Omron CX-Programmer project 疏蜞轳觇開钺祛蝼桕 (CX-Programmer 9.41)

# PLC 皖恹橄耸1: CP1E N40

## Global symbols (name address type ; comment)
0.00 BOOL  ; 原点接近
0.01 BOOL  ; 膜架上限
0.03 BOOL  ; 膜架下限
0.04 BOOL  ; 暂停
0.05 BOOL  ; 运行
0.06 BOOL  ; 急停
0.07 BOOL  ; 薄膜随动
0.08 BOOL  ; 减速接近
0.09 BOOL  ; 进料光电
0.11 BOOL  ; 货高与货到位光电
100.00 BOOL  ; 送膜转
100.01 BOOL  ; 模架下降
100.02 BOOL  ; 主机输送线转
100.04 BOOL  ; 转盘正传
100.05 BOOL  ; 转盘2段速
100.06 BOOL  ; 转盘3段速
100.07 BOOL  ; 膜架上升
101.00 BOOL  ; 夹膜
101.01 BOOL  ; 摆臂
101.02 BOOL  ; 断膜
101.03 BOOL  ; 扶膜
101.05 BOOL  ; 吹膜
101.07 BOOL  ; 送膜切换
102.04 BOOL  ; 压膜
102.05 BOOL  ; 吹摸
102.07 BOOL  ; 送膜切换
12.00 BOOL  ; 运行开始
12.01 BOOL  ; 进料光电触发位
12.02 BOOL  ; 触发运行延时
12.03 BOOL  ; 夹膜释放触发位
12.04 BOOL  ; 什么时候升到位
12.05 BOOL  ; 触发頂层计数
12.06 BOOL  ; 甚么时候下到位
12.07 BOOL  ; 底层技术开始
12.08 BOOL  ; 2段速进入位
12.09 BOOL  ; 2段速结束位
12.10 BOOL  ; 三段速进入位
12.11 BOOL  ; 停止位
12.12 BOOL  ; 摆臂触发位
12.13 BOOL  ; 触发出货
12.14 BOOL  ; 主机线停止
12.15 BOOL  ; 反复循环位
13.00 BOOL  ; 貨高光电触发位
13.01 BOOL  ; 停止膜上升
13.02 BOOL  ; 准备运行开始
13.03 BOOL  ; 运行准备完成
13.04 BOOL  ; 后送线停止
14.00 BOOL  ; 运行前回原点
14.01 BOOL  ; 运行前回下限位
15.00 BOOL  ; 包完后进3段速
15.01 BOOL  ; 包完后何时进3段速
1.00 BOOL  ; 出到位
1.01 BOOL  ; 货高与货到位光电
C001 BOOL  ; 减速计数
C002 BOOL  ; 底层设置数
C003 BOOL  ; 頂层计数
C004 BOOL  ; 往复次数设置数
C005 BOOL  ; 停止圈数
T010 BOOL  ; 运行延时
T011 BOOL  ; 货高延时
T012 BOOL  ; 压膜延时设置值
T013 BOOL  ; 夹膜设置值
T014 BOOL  ; 锻模设置值
T015 BOOL  ; 抚摸设置值
T016 BOOL  ; 出货设置值
T017 BOOL  ; 出货值加1
T018 BOOL  ; 吹膜延时
T100 BOOL  ; 货到延时
T200 BOOL  ; 模架下降延时
T202 BOOL  ; 落剪子延时
W10.00 BOOL  ; 手动后线转动
W10.01 BOOL  ; 模架上升触发位
W10.02 BOOL  ; 模架下降触发位
W10.03 BOOL  ; 主机输送线触发位
W10.04 BOOL  ; 手动夹膜
W10.05 BOOL  ; 手动转盘正传
W10.06 BOOL  ; 手动主机输送线转
W10.07 BOOL  ; 手动夹膜释放
W10.08 BOOL  ; 手动摆臂
W10.09 BOOL  ; 手动断膜
W10.10 BOOL  ; 手动抚摸
W10.11 BOOL  ; 手动膜架上升
W10.12 BOOL  ; 手动模架下降
W10.14 BOOL  ; 后线触发位
W10.15 BOOL  ; 手动压膜
W11.00 BOOL  ; 荚膜释放
W11.02 BOOL  ; 转盘正传触发位
W11.03 BOOL  ; 转盘2段速触发位
W11.04 BOOL  ; 转盘3段速触发位
W11.11 BOOL  ; 压膜
W11.12 BOOL  ; 锻模
W11.13 BOOL  ; 抚摸
W11.14 BOOL  ; 荚膜
W11.15 BOOL  ; 摆臂
W50.00 BOOL  ; 货到延时自锁
W80.00 BOOL  ; 夹膜释放
W80.01 BOOL  ; 荚膜
W80.02 BOOL  ; 吹膜

## Program 新程序1 (cyclic task 0)
Local symbols
好0 CHANNEL

### Section 段1

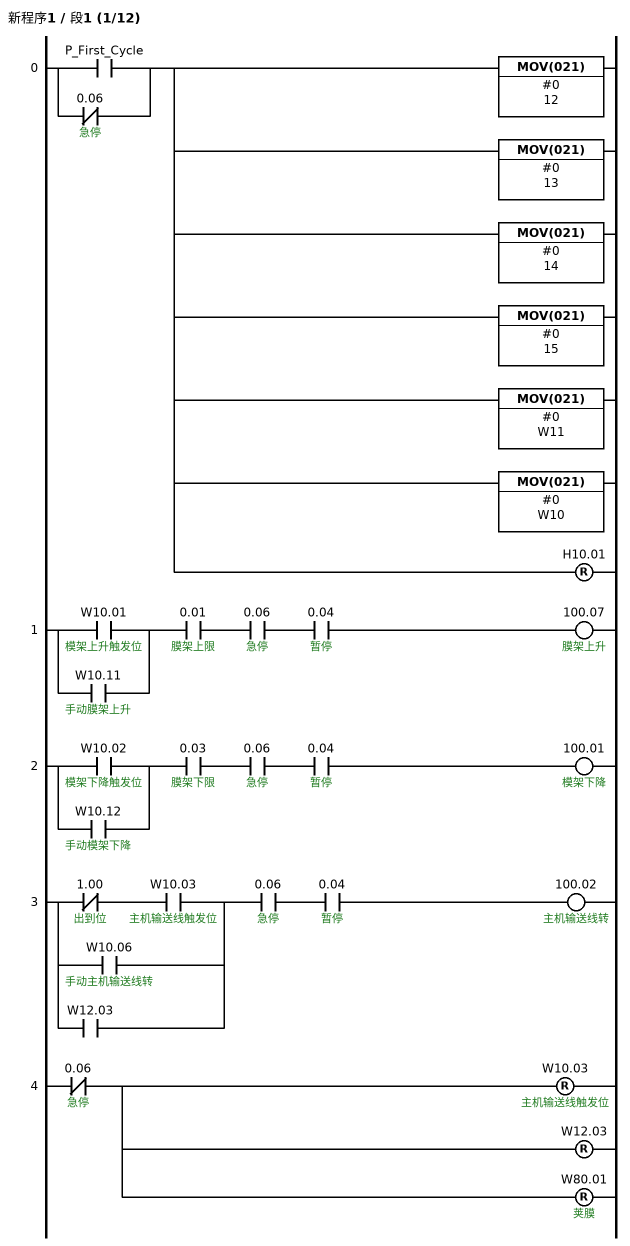
; rung 0
LD P_First_Cycle
ORNOT 0.06  ; 急停
MOV(021) #0 12
MOV(021) #0 13
MOV(021) #0 14
MOV(021) #0 15
MOV(021) #0 W11
MOV(021) #0 W10
RSET H10.01
; rung 1
LD W10.01  ; 模架上升触发位
OR W10.11  ; 手动膜架上升
AND 0.01  ; 膜架上限
AND 0.06  ; 急停
AND 0.04  ; 暂停
OUT 100.07  ; 膜架上升
; rung 2
LD W10.02  ; 模架下降触发位
OR W10.12  ; 手动模架下降
AND 0.03  ; 膜架下限
AND 0.06  ; 急停
AND 0.04  ; 暂停
OUT 100.01  ; 模架下降
; rung 3
LDNOT 1.00  ; 出到位
AND W10.03  ; 主机输送线触发位
OR W10.06  ; 手动主机输送线转
OR W12.03
AND 0.06  ; 急停
AND 0.04  ; 暂停
OUT 100.02  ; 主机输送线转
; rung 4
LDNOT 0.06  ; 急停
RSET W10.03  ; 主机输送线触发位
RSET W12.03
RSET W80.01  ; 荚膜

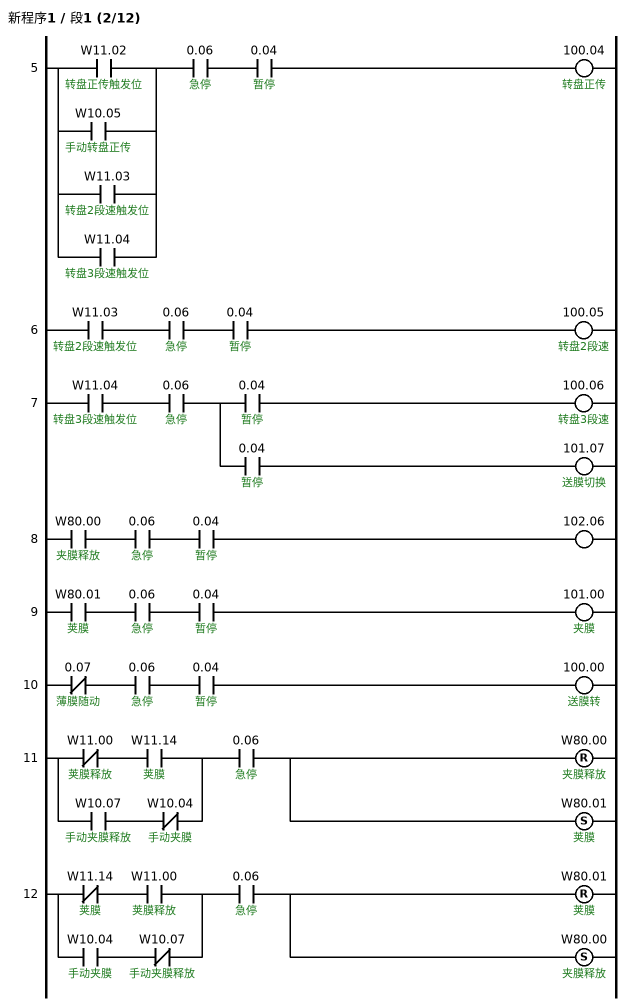
; rung 5
LD W11.02  ; 转盘正传触发位
OR W10.05  ; 手动转盘正传
OR W11.03  ; 转盘2段速触发位
OR W11.04  ; 转盘3段速触发位
AND 0.06  ; 急停
AND 0.04  ; 暂停
OUT 100.04  ; 转盘正传
; rung 6
LD W11.03  ; 转盘2段速触发位
AND 0.06  ; 急停
AND 0.04  ; 暂停
OUT 100.05  ; 转盘2段速
; rung 7
LD W11.04  ; 转盘3段速触发位
AND 0.06  ; 急停
OUT TR0
AND 0.04  ; 暂停
OUT 100.06  ; 转盘3段速
LD TR0
AND 0.04  ; 暂停
OUT 101.07  ; 送膜切换
; rung 8
LD W80.00  ; 夹膜释放
AND 0.06  ; 急停
AND 0.04  ; 暂停
OUT 102.06
; rung 9
LD W80.01  ; 荚膜
AND 0.06  ; 急停
AND 0.04  ; 暂停
OUT 101.00  ; 夹膜
; rung 10
LDNOT 0.07  ; 薄膜随动
AND 0.06  ; 急停
AND 0.04  ; 暂停
OUT 100.00  ; 送膜转
; rung 11
LDNOT W11.00  ; 荚膜释放
AND W11.14  ; 荚膜
LD W10.07  ; 手动夹膜释放
ANDNOT W10.04  ; 手动夹膜
ORLD
AND 0.06  ; 急停
RSET W80.00  ; 夹膜释放
SET W80.01  ; 荚膜
; rung 12
LDNOT W11.14  ; 荚膜
AND W11.00  ; 荚膜释放
LD W10.04  ; 手动夹膜
ANDNOT W10.07  ; 手动夹膜释放
ORLD
AND 0.06  ; 急停
RSET W80.01  ; 荚膜
SET W80.00  ; 夹膜释放

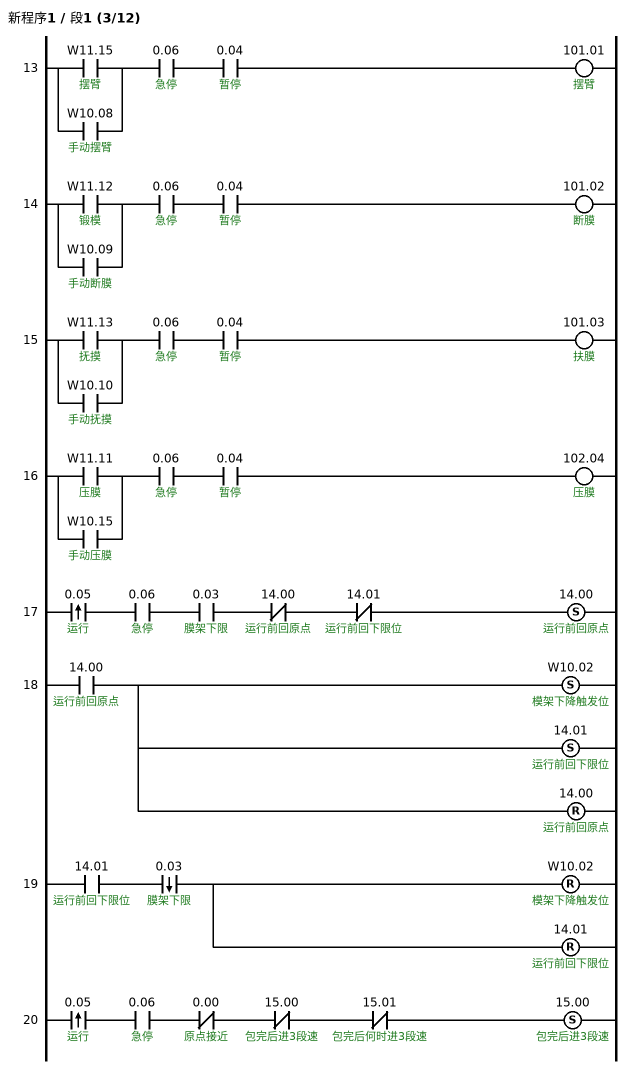
; rung 13
LD W11.15  ; 摆臂
OR W10.08  ; 手动摆臂
AND 0.06  ; 急停
AND 0.04  ; 暂停
OUT 101.01  ; 摆臂
; rung 14
LD W11.12  ; 锻模
OR W10.09  ; 手动断膜
AND 0.06  ; 急停
AND 0.04  ; 暂停
OUT 101.02  ; 断膜
; rung 15
LD W11.13  ; 抚摸
OR W10.10  ; 手动抚摸
AND 0.06  ; 急停
AND 0.04  ; 暂停
OUT 101.03  ; 扶膜
; rung 16
LD W11.11  ; 压膜
OR W10.15  ; 手动压膜
AND 0.06  ; 急停
AND 0.04  ; 暂停
OUT 102.04  ; 压膜
; rung 17
@LD 0.05  ; 运行
AND 0.06  ; 急停
AND 0.03  ; 膜架下限
ANDNOT 14.00  ; 运行前回原点
ANDNOT 14.01  ; 运行前回下限位
SET 14.00  ; 运行前回原点
; rung 18
LD 14.00  ; 运行前回原点
SET W10.02  ; 模架下降触发位
SET 14.01  ; 运行前回下限位
RSET 14.00  ; 运行前回原点
; rung 19
LD 14.01  ; 运行前回下限位
%AND 0.03  ; 膜架下限
RSET W10.02  ; 模架下降触发位
RSET 14.01  ; 运行前回下限位
; rung 20
@LD 0.05  ; 运行
AND 0.06  ; 急停
ANDNOT 0.00  ; 原点接近
ANDNOT 15.00  ; 包完后进3段速
ANDNOT 15.01  ; 包完后何时进3段速
SET 15.00  ; 包完后进3段速

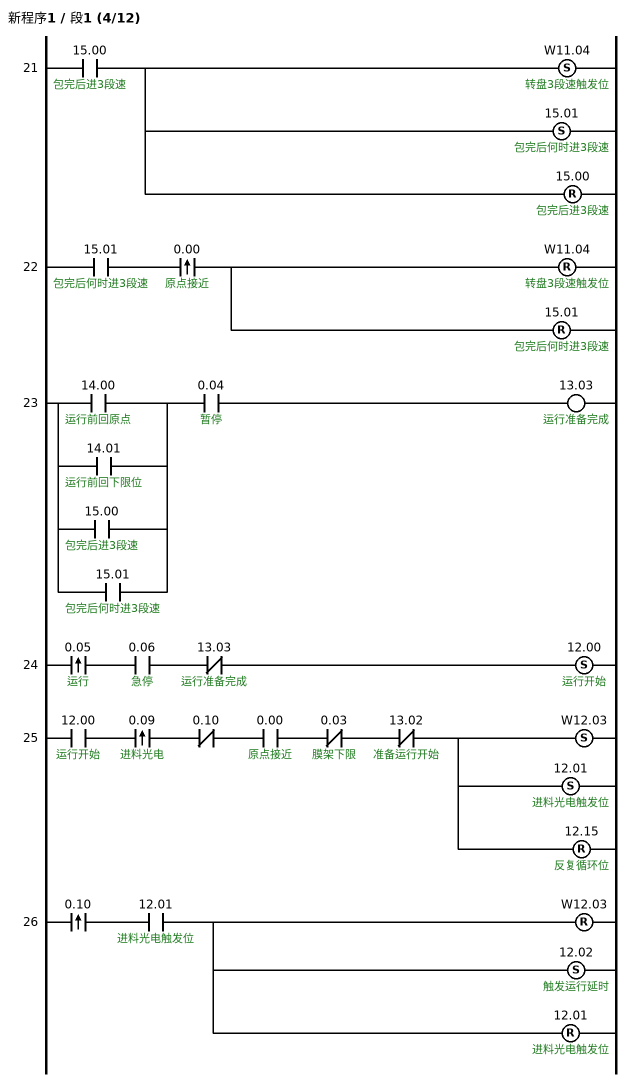
; rung 21
LD 15.00  ; 包完后进3段速
SET W11.04  ; 转盘3段速触发位
SET 15.01  ; 包完后何时进3段速
RSET 15.00  ; 包完后进3段速
; rung 22
LD 15.01  ; 包完后何时进3段速
@AND 0.00  ; 原点接近
RSET W11.04  ; 转盘3段速触发位
RSET 15.01  ; 包完后何时进3段速
; rung 23
LD 14.00  ; 运行前回原点
OR 14.01  ; 运行前回下限位
OR 15.00  ; 包完后进3段速
OR 15.01  ; 包完后何时进3段速
AND 0.04  ; 暂停
OUT 13.03  ; 运行准备完成
; rung 24
@LD 0.05  ; 运行
AND 0.06  ; 急停
ANDNOT 13.03  ; 运行准备完成
SET 12.00  ; 运行开始
; rung 25
LD 12.00  ; 运行开始
@AND 0.09  ; 进料光电
ANDNOT 0.10
AND 0.00  ; 原点接近
ANDNOT 0.03  ; 膜架下限
ANDNOT 13.02  ; 准备运行开始
SET W12.03
SET 12.01  ; 进料光电触发位
RSET 12.15  ; 反复循环位
; rung 26
@LD 0.10
AND 12.01  ; 进料光电触发位
RSET W12.03
SET 12.02  ; 触发运行延时
RSET 12.01  ; 进料光电触发位

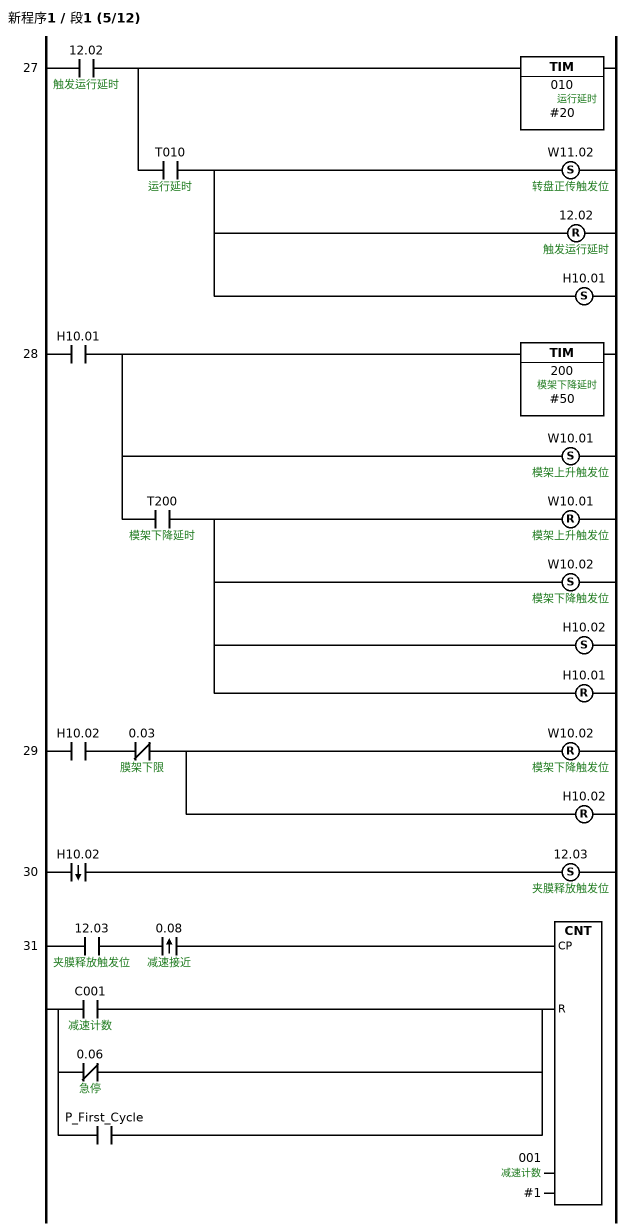
; rung 27
LD 12.02  ; 触发运行延时
TIM 010 #20  ; 运行延时
AND T010  ; 运行延时
SET W11.02  ; 转盘正传触发位
RSET 12.02  ; 触发运行延时
SET H10.01
; rung 28
LD H10.01
TIM 200 #50  ; 模架下降延时
SET W10.01  ; 模架上升触发位
AND T200  ; 模架下降延时
RSET W10.01  ; 模架上升触发位
SET W10.02  ; 模架下降触发位
SET H10.02
RSET H10.01
; rung 29
LD H10.02
ANDNOT 0.03  ; 膜架下限
RSET W10.02  ; 模架下降触发位
RSET H10.02
; rung 30
%LD H10.02
SET 12.03  ; 夹膜释放触发位
; rung 31
LD 12.03  ; 夹膜释放触发位
@AND 0.08  ; 减速接近
LD C001  ; 减速计数
ORNOT 0.06  ; 急停
OR P_First_Cycle
CNT 001 #1  ; 减速计数

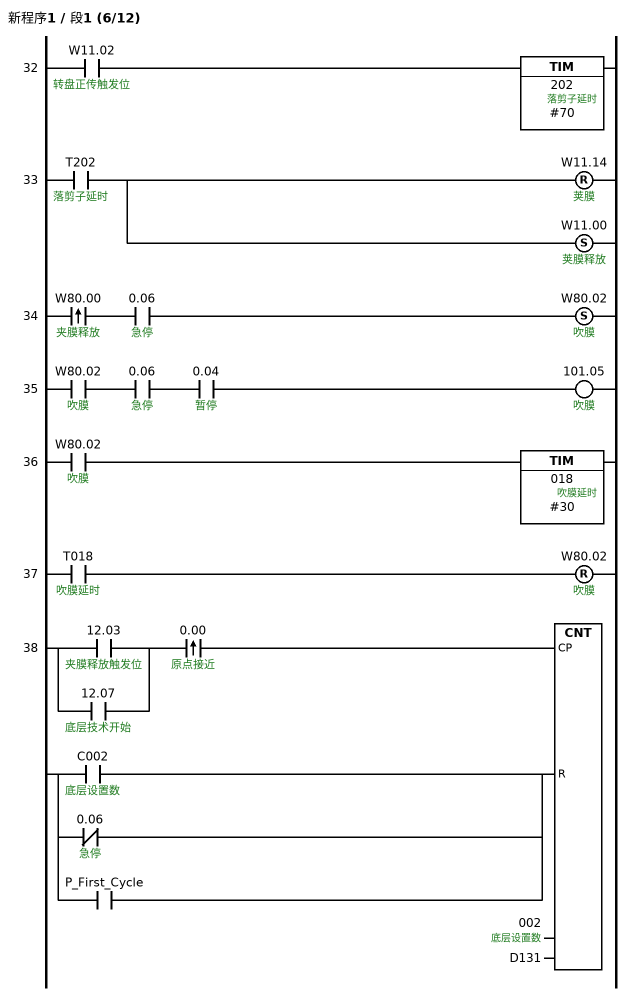
; rung 32
LD W11.02  ; 转盘正传触发位
TIM 202 #70  ; 落剪子延时
; rung 33
LD T202  ; 落剪子延时
RSET W11.14  ; 荚膜
SET W11.00  ; 荚膜释放
; rung 34
@LD W80.00  ; 夹膜释放
AND 0.06  ; 急停
SET W80.02  ; 吹膜
; rung 35
LD W80.02  ; 吹膜
AND 0.06  ; 急停
AND 0.04  ; 暂停
OUT 101.05  ; 吹膜
; rung 36
LD W80.02  ; 吹膜
TIM 018 #30  ; 吹膜延时
; rung 37
LD T018  ; 吹膜延时
RSET W80.02  ; 吹膜
; rung 38
LD 12.03  ; 夹膜释放触发位
OR 12.07  ; 底层技术开始
@AND 0.00  ; 原点接近
LD C002  ; 底层设置数
ORNOT 0.06  ; 急停
OR P_First_Cycle
CNT 002 D131  ; 底层设置数

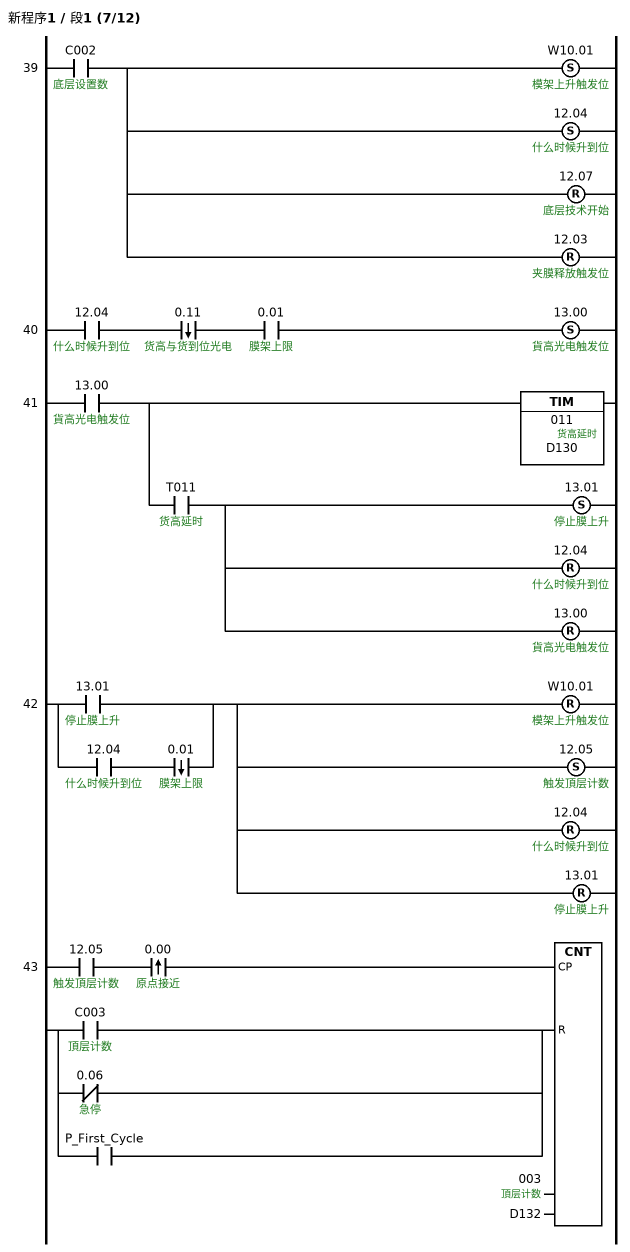
; rung 39
LD C002  ; 底层设置数
SET W10.01  ; 模架上升触发位
SET 12.04  ; 什么时候升到位
RSET 12.07  ; 底层技术开始
RSET 12.03  ; 夹膜释放触发位
; rung 40
LD 12.04  ; 什么时候升到位
%AND 0.11  ; 货高与货到位光电
AND 0.01  ; 膜架上限
SET 13.00  ; 貨高光电触发位
; rung 41
LD 13.00  ; 貨高光电触发位
TIM 011 D130  ; 货高延时
AND T011  ; 货高延时
SET 13.01  ; 停止膜上升
RSET 12.04  ; 什么时候升到位
RSET 13.00  ; 貨高光电触发位
; rung 42
LD 13.01  ; 停止膜上升
LD 12.04  ; 什么时候升到位
%AND 0.01  ; 膜架上限
ORLD
RSET W10.01  ; 模架上升触发位
SET 12.05  ; 触发頂层计数
RSET 12.04  ; 什么时候升到位
RSET 13.01  ; 停止膜上升
; rung 43
LD 12.05  ; 触发頂层计数
@AND 0.00  ; 原点接近
LD C003  ; 頂层计数
ORNOT 0.06  ; 急停
OR P_First_Cycle
CNT 003 D132  ; 頂层计数

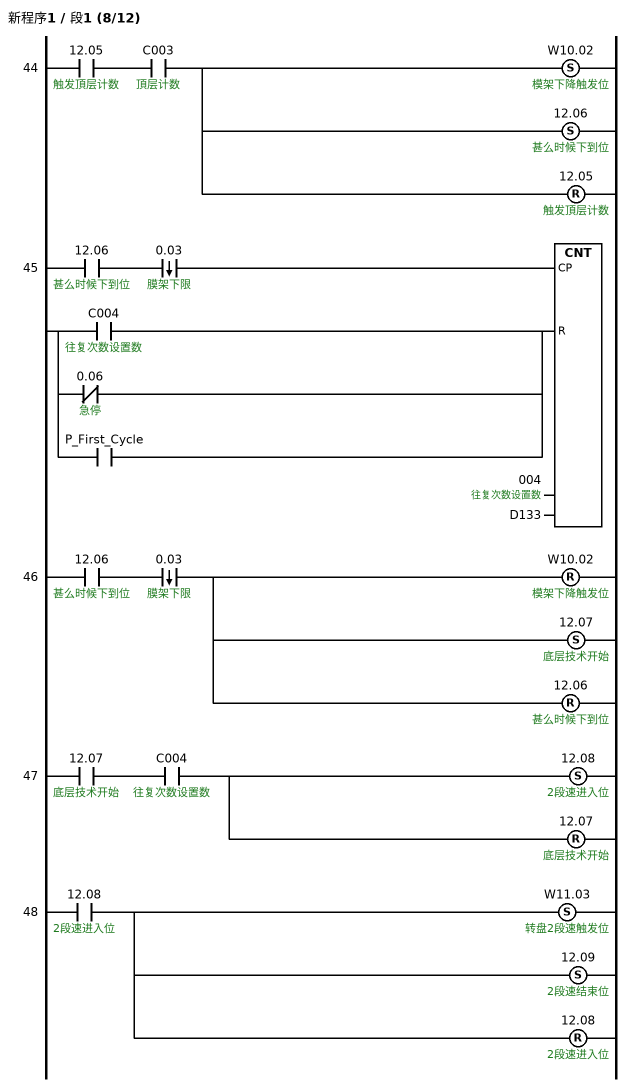
; rung 44
LD 12.05  ; 触发頂层计数
AND C003  ; 頂层计数
SET W10.02  ; 模架下降触发位
SET 12.06  ; 甚么时候下到位
RSET 12.05  ; 触发頂层计数
; rung 45
LD 12.06  ; 甚么时候下到位
%AND 0.03  ; 膜架下限
LD C004  ; 往复次数设置数
ORNOT 0.06  ; 急停
OR P_First_Cycle
CNT 004 D133  ; 往复次数设置数
; rung 46
LD 12.06  ; 甚么时候下到位
%AND 0.03  ; 膜架下限
RSET W10.02  ; 模架下降触发位
SET 12.07  ; 底层技术开始
RSET 12.06  ; 甚么时候下到位
; rung 47
LD 12.07  ; 底层技术开始
AND C004  ; 往复次数设置数
SET 12.08  ; 2段速进入位
RSET 12.07  ; 底层技术开始
; rung 48
LD 12.08  ; 2段速进入位
SET W11.03  ; 转盘2段速触发位
SET 12.09  ; 2段速结束位
RSET 12.08  ; 2段速进入位

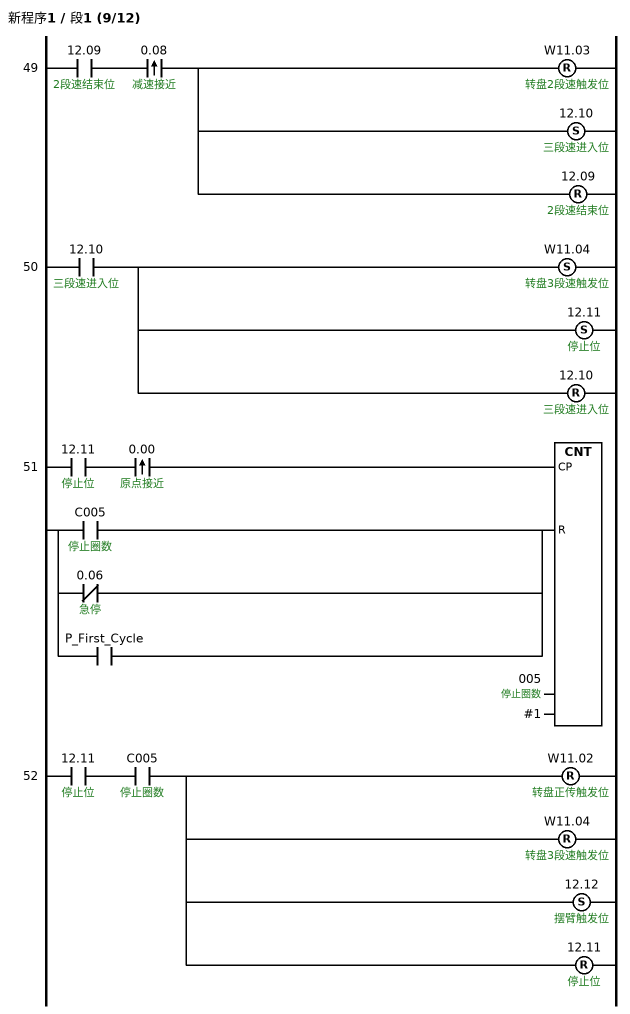
; rung 49
LD 12.09  ; 2段速结束位
@AND 0.08  ; 减速接近
RSET W11.03  ; 转盘2段速触发位
SET 12.10  ; 三段速进入位
RSET 12.09  ; 2段速结束位
; rung 50
LD 12.10  ; 三段速进入位
SET W11.04  ; 转盘3段速触发位
SET 12.11  ; 停止位
RSET 12.10  ; 三段速进入位
; rung 51
LD 12.11  ; 停止位
@AND 0.00  ; 原点接近
LD C005  ; 停止圈数
ORNOT 0.06  ; 急停
OR P_First_Cycle
CNT 005 #1  ; 停止圈数
; rung 52
LD 12.11  ; 停止位
AND C005  ; 停止圈数
RSET W11.02  ; 转盘正传触发位
RSET W11.04  ; 转盘3段速触发位
SET 12.12  ; 摆臂触发位
RSET 12.11  ; 停止位

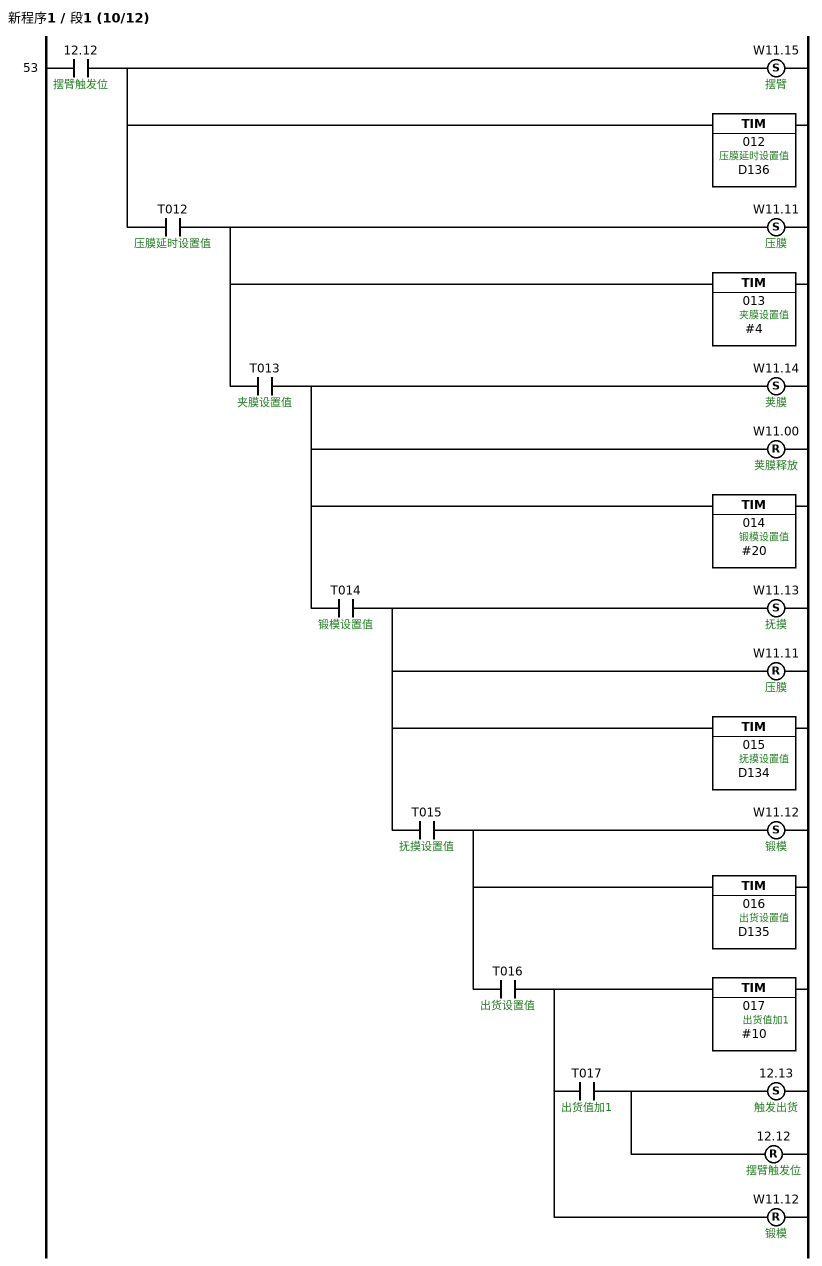
; rung 53
LD 12.12  ; 摆臂触发位
SET W11.15  ; 摆臂
TIM 012 D136  ; 压膜延时设置值
AND T012  ; 压膜延时设置值
SET W11.11  ; 压膜
TIM 013 #4  ; 夹膜设置值
AND T013  ; 夹膜设置值
SET W11.14  ; 荚膜
RSET W11.00  ; 荚膜释放
TIM 014 #20  ; 锻模设置值
AND T014  ; 锻模设置值
SET W11.13  ; 抚摸
RSET W11.11  ; 压膜
TIM 015 D134  ; 抚摸设置值
AND T015  ; 抚摸设置值
SET W11.12  ; 锻模
TIM 016 D135  ; 出货设置值
AND T016  ; 出货设置值
OUT TR0
TIM 017 #10  ; 出货值加1
AND T017  ; 出货值加1
SET 12.13  ; 触发出货
RSET 12.12  ; 摆臂触发位
LD TR0
RSET W11.12  ; 锻模

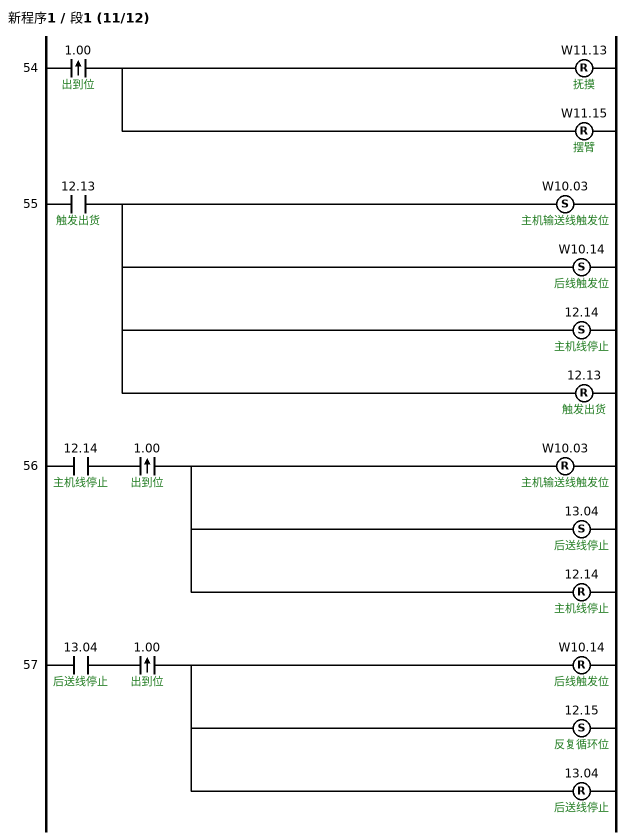
; rung 54
@LD 1.00  ; 出到位
RSET W11.13  ; 抚摸
RSET W11.15  ; 摆臂
; rung 55
LD 12.13  ; 触发出货
SET W10.03  ; 主机输送线触发位
SET W10.14  ; 后线触发位
SET 12.14  ; 主机线停止
RSET 12.13  ; 触发出货
; rung 56
LD 12.14  ; 主机线停止
@AND 1.00  ; 出到位
RSET W10.03  ; 主机输送线触发位
SET 13.04  ; 后送线停止
RSET 12.14  ; 主机线停止
; rung 57
LD 13.04  ; 后送线停止
@AND 1.00  ; 出到位
RSET W10.14  ; 后线触发位
SET 12.15  ; 反复循环位
RSET 13.04  ; 后送线停止

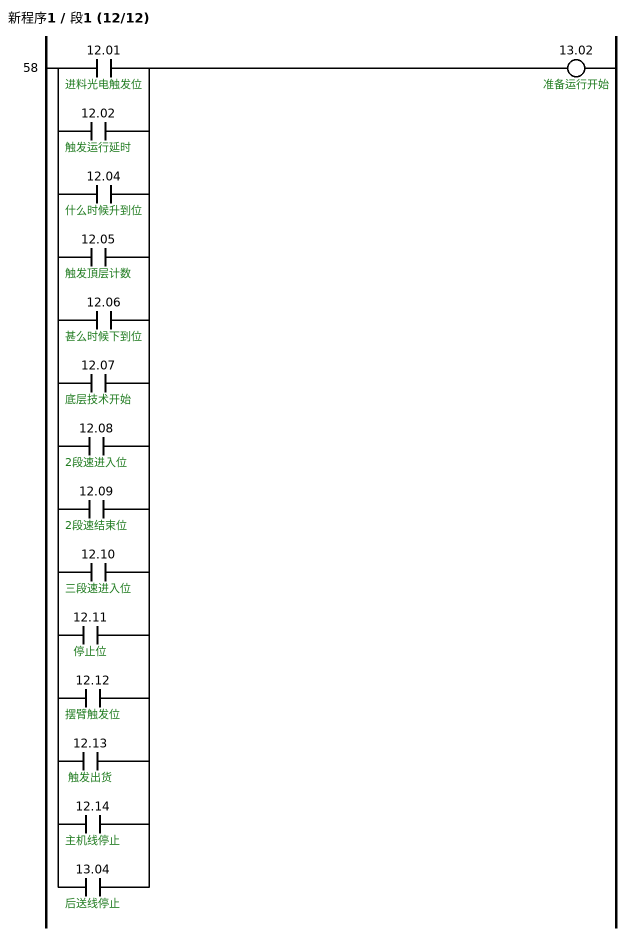
; rung 58
LD 12.01  ; 进料光电触发位
OR 12.02  ; 触发运行延时
OR 12.04  ; 什么时候升到位
OR 12.05  ; 触发頂层计数
OR 12.06  ; 甚么时候下到位
OR 12.07  ; 底层技术开始
OR 12.08  ; 2段速进入位
OR 12.09  ; 2段速结束位
OR 12.10  ; 三段速进入位
OR 12.11  ; 停止位
OR 12.12  ; 摆臂触发位
OR 12.13  ; 触发出货
OR 12.14  ; 主机线停止
OR 13.04  ; 后送线停止
OUT 13.02  ; 准备运行开始

### Section 段2
; rung 0
END(001)